TYPE STATE:
    STRUCT
        curTime: REAL;
        dvar_M_g2_aut_z: DINT;
    END_STRUCT;
END_TYPE
